Staubli VAL3: stop.pgx

program stop()
begin


end
